Staubli VAL3: onRightEvent.pgx

program onRightEvent()
begin
  call save:FwdBoxType()
  call buildList()
end
